(* IEC 61131-3 sources: TIAX_Demo/src, 2 files *)

(* ---- library.st ---- *)
NAMESPACE MotorLibrary

    CLASS PUBLIC Motor
        VAR PRIVATE
            _started : BOOL;
        END_VAR

        VAR PRIVATE

        END_VAR

        METHOD PUBLIC Start : BOOL
            _started := TRUE;
            Start := TRUE;
        END_METHOD

        METHOD PUBLIC Stop : BOOL
            _started := FALSE;
            Stop := TRUE;
        END_METHOD

    END_CLASS

END_NAMESPACE

(* ---- wrapper.st ---- *)
NAMESPACE MotorLibrary

    FUNCTION_BLOCK MotorWrapper
        VAR_INPUT
            start   : BOOL;
            stop    : BOOL;
        END_VAR
       VAR_OUTPUT
            Inmotion: BOOL; (* fornuftig kommentar *)
       END_VAR

        VAR
            m : Motor;
        END_VAR

        IF start THEN
            m.Start();
            Inmotion := TRUE;
        END_IF;

        IF stop THEN
            m.Stop();
            Inmotion := FALSE;
        END_IF;

    END_FUNCTION_BLOCK

END_NAMESPACE
